FUNCTION_BLOCK AirPiston
VAR_INPUT CONSTANT
	bEnable : BOOL;
END_VAR
VAR_OUTPUT
	valveIn AT %Q* : BOOL;
	valveOut AT %Q* : BOOL;
	
	contact AT %I* : BOOL;
	
	home AT %I* : BOOL;
	innerLimit AT %I* : BOOL;
	
	ready : BOOL;
	busy : BOOL;
	error : BOOL;
	homeSet : BOOL;
END_VAR
VAR
	reversalBrakeTrig : R_TRIG;
	
	step : Homing;
	mode : (HOLD, IN, OUT);
END_VAR

IF NOT bEnable THEN
	valveIn := FALSE;
	valveOut := FALSE;
	RETURN;
END_IF

IF home OR innerLimit THEN
	mode := HOLD;
END_IF

reversalBrakeTrig(CLK:= , Q=> valveOut); //short brake, Q does not change until the scan after CLK is set
reversalBrakeTrig.CLK := FALSE;

CASE mode OF
	HOLD:
		valveIn := FALSE;
		valveOut := FALSE;
		
	IN:
		valveIn := TRUE;
		valveOut := FALSE;
		
		IF reversalBrakeTrig.Q THEN //brake triggered
			mode := HOLD;
			
		ELSIF contact THEN
			valveIn := FALSE;
			reversalBrakeTrig.CLK := TRUE; //trigger brake
		END_IF
		
	OUT:
		valveIn := FALSE;
		valveOut := TRUE;
		
END_CASE

METHOD homingSequence : BOOL
(*
this version of homing always traverses to the inner limit before returning to home,
eliminating the possibility of reaching the outer limit while homing
*)
CASE step OF
	Homing.IDLE:
		step := Homing.OUT;
		
	Homing.OUT: //towards home
		mode := OUT;
		
		IF home THEN //if reached home
			step := Homing.DONE;
		END_IF
		
	Homing.DONE:
		mode := HOLD;
		homeSet := TRUE;
		
		homingSequence := TRUE;		
	
END_CASE
END_METHOD

METHOD slideIn : BOOL
VAR_INPUT
END_VAR
mode := IN;

slideIn := TRUE;
END_METHOD

METHOD slideOut : BOOL
VAR_INPUT
END_VAR
mode := OUT;

slideOut := TRUE;
END_METHOD

METHOD stop : BOOL
VAR_INPUT
END_VAR
valveIn := FALSE;
valveOut := FALSE;
mode := HOLD;

stop := TRUE;
END_METHOD

END_FUNCTION_BLOCK

(* stored: Version 1.1.0.1, ProductVersion 3.1.4024.11
   POU AirPiston: Id {ef8d0471-4ac2-4d12-9e08-c4e8a3719cb6}, SpecialFunc None
   Method homingSequence: Id {c3ff30f8-ced2-4f8e-b758-e21ca109ec69}
   Method slideIn: Id {c905417d-ebb0-4426-b712-8b35f4512697}
   Method slideOut: Id {d6cfbb92-1846-4f17-b88f-dcdab10c19f1}
   Method stop: Id {c035c442-83bc-4f21-a06c-19730e7f9f48} *)
